PROGRAM MAIN
VAR
	fbMarquee		:FB_Marquee;
	bLamp01,bLamp02,bLamp03,bLamp04		:BOOL;
	bBlinking			:BOOL;
	
	fbMarqueeEx		:FB_MarqueeEx;
	tDelay			:TIME:=T#500MS;
	
	
	fbMarqueeExPause		:FB_MarqueeExPause;
	bPause					:BOOL;
	bStop					:BOOL;
END_VAR

//==========Test FB_Marquee===========
//fbMarquee(pLamp01:= ADR(bLamp01) , pLamp02:=ADR(bLamp02), pLamp03:=ADR(bLamp03) , pLamp04:= ADR(bLamp04));
//fbMarquee.Blinking(bStart :=bBlinking );
//==========Test FB_Marquee===========


//===============Test FB_MarqueeEx======================
//fbMarqueeEx(pLamp01:= ADR(bLamp01) , pLamp02:=ADR(bLamp02),
//			 pLamp03:=ADR(bLamp03) , pLamp04:= ADR(bLamp04),pTime:= ADR(tDelay));
			 
//fbMarqueeEx.Blinking(bStart := bBlinking);
//===============Test FB_MarqueeEx======================


//===============Test FB_MarqueeExPause======================
(*fbMarqueeExPause(pLamp01:= ADR(bLamp01) , pLamp02:=ADR(bLamp02),
			 pLamp03:=ADR(bLamp03) , pLamp04:= ADR(bLamp04),pTime:= ADR(tDelay),pPause:= ADR(bPause),pStop := ADR(bStop));
fbMarqueeExPause.Blinking(bStart :=bBlinking);  *)

END_PROGRAM

(* stored: Version 1.1.0.1, ProductVersion 3.1.4022.16
   POU MAIN: Id {fa671d83-edd0-492d-886f-c7d702fe85de}, SpecialFunc None *)
